FUNCTION_BLOCK FB_Modbus_Send_FIFO
VAR_INPUT
	stInput				:ST_Modbus_Send_Frame;
END_VAR
VAR_OUTPUT
	bExistMessage		:BOOL;
	nBufferCount		:UDINT;
	nLoad				:REAL;
	stOutput			:ST_Modbus_Send_Frame;
END_VAR
VAR
	ArrBuffer			:ARRAY[0..10000] OF BYTE;
	fbBuffer			:FB_MemRingBuffer;
	bOk					:BOOL;
	cbSize				:UDINT;
	
	nCurrentBuffer		:UDINT;
	BufferSize			:UINT;
END_VAR

bExistMessage := nBufferCount > 0;
BufferSize := SIZEOF(ArrBuffer);
nLoad :=  (UDINT_TO_REAL(fbBuffer.cbSize)/UDINT_TO_REAL(BufferSize)) * 100.0;;

ACTION A_Add:
fbBuffer.A_AddTail(	pWrite:=ADR(stInput),
					cbWrite:= SIZEOF( stInput ),
					pBuffer:= ADR( arrBuffer ),
					cbBuffer:= SIZEOF( arrBuffer ),
					bOk=> bOk,
					nCount => nBufferCount );
END_ACTION

ACTION A_Remove:
fbBuffer.A_RemoveHead(
						pRead:= ADR(stOutput ),
						cbRead:= SIZEOF( stOutput ),
						pBuffer:= ADR( arrBuffer ),
						cbBuffer:= SIZEOF( arrBuffer ),
						bOk=> bOk,
						nCount => nBufferCount );
END_ACTION

ACTION A_Reset:
MEMSET(ADR(ArrBuffer),0,SIZEOF(ArrBuffer));

fbBuffer.A_Reset(bOk=>bOk,
			nCount=>nBufferCount);			
			bExistMessage := nBufferCount > 0;
nLoad := fbBuffer.cbSize  / 200;
END_ACTION

END_FUNCTION_BLOCK

(* stored: Version 1.1.0.1
   POU FB_Modbus_Send_FIFO: Id {971fcccc-f3d5-45f2-9d7f-e73bbf056593}, SpecialFunc None
   Action A_Add: Id {9d978233-6a95-46db-873c-61b12168c27b}
   Action A_Remove: Id {4d04fd7d-30d2-42f4-be48-5ee41b38f025}
   Action A_Reset: Id {ba558b3d-19c3-45d2-b0f7-2fba583faf71} *)
